// TIA Portal V17 export
// export: Created 2024-08-26T21:07:15.6305429Z, ExportSetting WithDefaults, DisplayName Totally Integrated Automation Portal, DisplayVersion V17 Update 7, DisplayName TIA Portal Openness, DisplayVersion V17 Update 7, DisplayName TIA Portal Version Control Interface, DisplayVersion V17, DisplayName SINAMICS Startdrive Advanced, DisplayVersion V17 SP2, DisplayName SINAMICS Startdrive G110M, G120, G120C, G120D, G120P, G115D, DisplayVersion V17 SP2, DisplayName SINAMICS Startdrive G130, G150, S120, S150, SINAMICS MV, S210, DisplayVersion V17 SP2, DisplayName STEP 7 Professional, DisplayVersion V17 Update 7, DisplayName STEP 7 Safety, DisplayVersion V17 Update 6, DisplayName WinCC Advanced / Unified PC, DisplayVersion V17 Update 7
DATA_BLOCK "DB_INPUTS"   // DB1
{ S7_Optimized_Access := 'TRUE' }
VERSION : 0.1
// stored: AutoNumber false, DBAccessibleFromOPCUA true, DBAccessibleFromWebserver true, IsOnlyStoredInLoadMemory false, IsRetainMemResEnabled false, IsWriteProtectedInAS false, MemoryReserve 100
   VAR RETAIN
      intputSequence : Array[0..32, 0..25] of DInt;   // 32 entradas [modelo, paso]
   END_VAR
   VAR
      activeInputsReq : Array[0..31] of Bool;
   END_VAR
   VAR RETAIN
      maskSequence : Array[0..32, 0..25] of DInt;   // Máscara de entradas
   END_VAR
   VAR
      activeMask : Array[0..31] of Bool;
   END_VAR
   VAR RETAIN
      inputText : Array[0..31] of String;   // Texto HMI de cada entrada
   END_VAR
   VAR
      buttonStatus : Array[0..63] of Bool;
      activeInputsReqDInt : DInt := -2_130_444_284;   // Estado de sensores en directo
      inputActive : Array[0..31] of Bool;
      euchnerReading : Array[0..254] of Char;
      nestScannerReading : String := '';
      upperScannerReading : String := '';
      nestScanerReceived : Array[0..254] of Char;
      nestScanerReceivedString : String := '';
      upperScannerReceived : Array[0..254] of Char;
      upperScannerReceivedString : String := '';
      euchnerReadingString : String := '$01';
      laserReading : Word := 16#0000;
      laserConstant : Real := 0.0005802801;
      laserReadingInt : DInt := 0;
      readingConversion : LReal := 0.0;
      euchnerName : String := '';
      euchner : Array[0..257] of Byte;
   END_VAR
BEGIN
   intputSequence[0,0] := -2_130_444_283;
   intputSequence[0,1] := -1_996_150_012;
   intputSequence[0,2..4] := -2_146_096_376;
   intputSequence[0,5] := -2_130_367_736;
   intputSequence[0,6..7] := -2_130_367_740;
   intputSequence[0,8] := -2_130_444_284;
   intputSequence[0,9..25] := 0;
   intputSequence[1,0] := -2_130_444_283;
   intputSequence[1,1] := -1_996_082_428;
   intputSequence[1,2..3] := -2_142_358_768;
   intputSequence[1,4] := -2_142_358_640;
   intputSequence[1,5] := -2_142_358_652;
   intputSequence[1,6..7] := -2_130_300_156;
   intputSequence[1,8] := -2_130_444_284;
   intputSequence[1,9..25] := 0;
   intputSequence[2,0] := -2_130_444_283;
   intputSequence[2,1] := -1_996_150_012;
   intputSequence[2,2..4] := -2_146_096_376;
   intputSequence[2,5] := -2_130_367_736;
   intputSequence[2,6..7] := -2_130_367_740;
   intputSequence[2,8] := -2_130_444_284;
   intputSequence[2,9..25] := 0;
   intputSequence[3,0] := 84148229;
   intputSequence[3,1] := 1_057_235_716;
   intputSequence[3,2] := 1_175_724_802;
   intputSequence[3,3] := 101_720_834;
   intputSequence[3,4] := 101_982_978;
   intputSequence[3,5] := 84157188;
   intputSequence[3,6] := 84148228;
   intputSequence[3,7..25] := 0;
   intputSequence[4,0] := 84148229;
   intputSequence[4,1] := 1_057_236_740;
   intputSequence[4,2] := 1_175_725_826;
   intputSequence[4,3] := 101_721_858;
   intputSequence[4,4] := 101_984_002;
   intputSequence[4,5] := 84158212;
   intputSequence[4,6] := 84148228;
   intputSequence[4,7..25] := 0;
   intputSequence[5,0] := 84148229;
   intputSequence[5,1] := 1_057_284_868;
   intputSequence[5,2] := 1_175_773_954;
   intputSequence[5,3] := 101_769_986;
   intputSequence[5,4] := 102_032_130;
   intputSequence[5,5] := 84206340;
   intputSequence[5,6] := 84148228;
   intputSequence[5,7..25] := 0;
   intputSequence[6,0] := 84148229;
   intputSequence[6,1] := 1_057_285_892;
   intputSequence[6,2] := 1_175_774_978;
   intputSequence[6,3] := 101_771_010;
   intputSequence[6,4] := 102_033_154;
   intputSequence[6,5] := 84207364;
   intputSequence[6,6] := 84148228;
   intputSequence[6,7..25] := 0;
   intputSequence[7,0] := 23724868;
   intputSequence[7,1] := 827_780_422;
   intputSequence[7,2] := 44756294;
   intputSequence[7,3] := 44755974;
   intputSequence[7,4] := 1_252_650_334;
   intputSequence[7,5..7] := 1_118_432_670;
   intputSequence[7,8] := 1_118_432_414;
   intputSequence[7,9] := 44630336;
   intputSequence[7,10..25] := 0;
   intputSequence[8,0] := 23724353;
   intputSequence[8,1] := 827_776_326;
   intputSequence[8,2] := 44752198;
   intputSequence[8,3] := 44751878;
   intputSequence[8,4] := 1_252_646_238;
   intputSequence[8,5] := 1_118_428_574;
   intputSequence[8,6] := 1_118_428_318;
   intputSequence[8,7] := 1_118_428_574;
   intputSequence[8,8] := 1_118_428_318;
   intputSequence[8,9] := 44630336;
   intputSequence[8,10..25] := 0;
   intputSequence[9,0] := 321;
   intputSequence[9,1] := 4193656;
   intputSequence[9,2] := 2_017_459_576;
   intputSequence[9,3] := 1_077_935_482;
   intputSequence[9,4] := 1_073_745_282;
   intputSequence[9,5..6] := 1_073_745_538;
   intputSequence[9,7..9] := 320;
   intputSequence[9,10..25] := 0;
   intputSequence[10,0] := 321;
   intputSequence[10,1] := 4193656;
   intputSequence[10,2] := 2_017_459_576;
   intputSequence[10,3] := 1_077_935_482;
   intputSequence[10,4] := 1_073_745_282;
   intputSequence[10,5..6] := 1_073_745_538;
   intputSequence[10,7..9] := 320;
   intputSequence[10,10..25] := 0;
   intputSequence[11,0] := 321;
   intputSequence[11,1] := 4193656;
   intputSequence[11,2] := 2_017_459_576;
   intputSequence[11,3] := 1_077_935_482;
   intputSequence[11,4] := 1_073_745_282;
   intputSequence[11,5..6] := 1_073_745_538;
   intputSequence[11,7..9] := 320;
   intputSequence[11,10..25] := 0;
   intputSequence[12,0] := 321;
   intputSequence[12,1] := 8387960;
   intputSequence[12,2] := 2_021_653_880;
   intputSequence[12,3] := 1_082_129_786;
   intputSequence[12,4] := 1_077_939_586;
   intputSequence[12,5] := 1_077_939_842;
   intputSequence[12,6] := 1_073_745_538;
   intputSequence[12,7..9] := 320;
   intputSequence[12,10..25] := 0;
   intputSequence[13,0] := 321;
   intputSequence[13,1] := 4193656;
   intputSequence[13,2] := 2_017_459_576;
   intputSequence[13,3] := 1_077_935_482;
   intputSequence[13,4] := 1_073_745_282;
   intputSequence[13,5..6] := 1_073_745_538;
   intputSequence[13,7..9] := 320;
   intputSequence[13,10..25] := 0;
   intputSequence[14,0] := 321;
   intputSequence[14,1] := 4193656;
   intputSequence[14,2] := 2_017_459_576;
   intputSequence[14,3] := 1_077_935_482;
   intputSequence[14,4] := 1_073_745_282;
   intputSequence[14,5..6] := 1_073_745_538;
   intputSequence[14,7..9] := 320;
   intputSequence[14,10..25] := 0;
   intputSequence[15,0] := 11;
   intputSequence[15,1] := 63040522;
   intputSequence[15,2] := 1_338_108_938;
   intputSequence[15,3] := 65137674;
   intputSequence[15,4] := 65135628;
   intputSequence[15,5] := 65134612;
   intputSequence[15,6] := 57344;
   intputSequence[15,7] := 805_363_712;
   intputSequence[15,8] := 10;
   intputSequence[15,9..25] := 0;
   intputSequence[16,0] := 321;
   intputSequence[16,1] := 8387960;
   intputSequence[16,2] := 2_021_653_880;
   intputSequence[16,3] := 1_082_129_786;
   intputSequence[16,4] := 1_077_939_586;
   intputSequence[16,5] := 1_077_939_842;
   intputSequence[16,6] := 1_073_745_538;
   intputSequence[16,7..9] := 320;
   intputSequence[16,10..25] := 0;
   intputSequence[17,0] := 321;
   intputSequence[17,1] := 4193656;
   intputSequence[17,2] := 2_017_459_576;
   intputSequence[17,3] := 1_077_935_482;
   intputSequence[17,4] := 1_073_745_282;
   intputSequence[17,5..6] := 1_073_745_538;
   intputSequence[17,7..9] := 320;
   intputSequence[17,10..25] := 0;
   intputSequence[18,0] := 321;
   intputSequence[18,1] := 4193656;
   intputSequence[18,2] := 2_017_459_576;
   intputSequence[18,3] := 1_077_935_482;
   intputSequence[18,4] := 1_073_745_282;
   intputSequence[18,5..6] := 1_073_745_538;
   intputSequence[18,7..9] := 320;
   intputSequence[18,10..25] := 0;
   intputSequence[19,0] := 321;
   intputSequence[19,1] := 4193656;
   intputSequence[19,2] := 2_017_459_576;
   intputSequence[19,3] := 1_077_935_482;
   intputSequence[19,4] := 1_073_745_282;
   intputSequence[19,5..6] := 1_073_745_538;
   intputSequence[19,7..9] := 320;
   intputSequence[19,10..25] := 0;
   intputSequence[20,0..25] := 0;
   intputSequence[21,0..25] := 0;
   intputSequence[22,0..25] := 0;
   intputSequence[23,0..25] := 0;
   intputSequence[24,0..25] := 0;
   intputSequence[25,0..25] := 0;
   intputSequence[26,0..25] := 0;
   intputSequence[27,0..25] := 0;
   intputSequence[28,0..25] := 0;
   intputSequence[29,0..25] := 0;
   intputSequence[30,0..25] := 0;
   intputSequence[31,0..25] := 0;
   intputSequence[32,0..25] := 0;
   activeInputsReq[0] := TRUE;
   activeInputsReq[1] := FALSE;
   activeInputsReq[2] := TRUE;
   activeInputsReq[3..17] := FALSE;
   activeInputsReq[18] := TRUE;
   activeInputsReq[19..23] := FALSE;
   activeInputsReq[24] := TRUE;
   activeInputsReq[25..30] := FALSE;
   activeInputsReq[31] := TRUE;
   maskSequence[0,0] := 0;
   maskSequence[0,1] := 805_306_368;
   maskSequence[0,2] := 939_528_320;
   maskSequence[0,3] := 134_221_952;
   maskSequence[0,4] := 146_804_928;
   maskSequence[0,5] := 134_217_856;
   maskSequence[0,6..8] := 134_217_728;
   maskSequence[0,9..25] := 0;
   maskSequence[1,0] := 0;
   maskSequence[1,1] := 805_306_368;
   maskSequence[1,2] := 939_526_144;
   maskSequence[1,3..4] := 134_219_776;
   maskSequence[1,5] := 138_412_160;
   maskSequence[1,6] := 134_221_952;
   maskSequence[1,7..8] := 134_217_728;
   maskSequence[1,9..25] := 0;
   maskSequence[2,0] := 0;
   maskSequence[2,1] := 805_306_368;
   maskSequence[2,2] := 939_528_320;
   maskSequence[2,3] := 134_221_952;
   maskSequence[2,4] := 146_804_928;
   maskSequence[2,5] := 134_217_856;
   maskSequence[2,6..8] := 134_217_728;
   maskSequence[2,9..25] := 0;
   maskSequence[3,0] := 0;
   maskSequence[3,1] := 202752;
   maskSequence[3,2] := 948_115_456;
   maskSequence[3,3] := 2_055_411_712;
   maskSequence[3,4] := 998_447_104;
   maskSequence[3,5] := 948_115_456;
   maskSequence[3,6] := 939_726_848;
   maskSequence[3,7..25] := 0;
   maskSequence[4,0] := 0;
   maskSequence[4,1] := 202752;
   maskSequence[4,2] := 948_115_456;
   maskSequence[4,3] := 2_055_411_712;
   maskSequence[4,4] := 998_447_104;
   maskSequence[4,5] := 948_115_456;
   maskSequence[4,6] := 939_726_848;
   maskSequence[4,7..25] := 0;
   maskSequence[5,0] := 0;
   maskSequence[5,1] := 202752;
   maskSequence[5,2] := 948_115_456;
   maskSequence[5,3] := 2_055_411_712;
   maskSequence[5,4] := 998_447_104;
   maskSequence[5,5] := 948_115_456;
   maskSequence[5,6] := 939_726_848;
   maskSequence[5,7..25] := 0;
   maskSequence[6,0] := 0;
   maskSequence[6,1] := 202752;
   maskSequence[6,2] := 948_115_456;
   maskSequence[6,3] := 2_055_411_712;
   maskSequence[6,4] := 998_447_104;
   maskSequence[6,5] := 948_115_456;
   maskSequence[6,6] := 939_726_848;
   maskSequence[6,7..25] := 0;
   maskSequence[7,0] := 66848767;
   maskSequence[7,1] := 66846720;
   maskSequence[7,2..3] := 66847168;
   maskSequence[7,4..6] := 66846720;
   maskSequence[7,7] := 66846976;
   maskSequence[7,8] := 66846720;
   maskSequence[7,9] := 66847168;
   maskSequence[7,10..25] := 0;
   maskSequence[8,0..1] := 66846720;
   maskSequence[8,2..3] := 66847168;
   maskSequence[8,4..5] := 66846720;
   maskSequence[8,6..7] := 66846976;
   maskSequence[8,8] := 66846720;
   maskSequence[8,9] := 66847168;
   maskSequence[8,10..25] := 0;
   maskSequence[9,0] := -322;
   maskSequence[9,1] := 2_014_248_960;
   maskSequence[9,2..3] := 983040;
   maskSequence[9,4..5] := 79687736;
   maskSequence[9,6] := 134_213_948;
   maskSequence[9,7..8] := -2;
   maskSequence[9,9] := 134_217_406;
   maskSequence[9,10..25] := 0;
   maskSequence[10,0] := -322;
   maskSequence[10,1] := 2_014_289_920;
   maskSequence[10,2..3] := 1024000;
   maskSequence[10,4..5] := 79687736;
   maskSequence[10,6] := 134_213_948;
   maskSequence[10,7..8] := -2;
   maskSequence[10,9] := 134_217_406;
   maskSequence[10,10..25] := 0;
   maskSequence[11,0] := -322;
   maskSequence[11,1] := 2_014_248_960;
   maskSequence[11,2..3] := 983040;
   maskSequence[11,4..5] := 79687736;
   maskSequence[11,6] := 134_213_948;
   maskSequence[11,7..8] := -2;
   maskSequence[11,9] := 134_217_406;
   maskSequence[11,10..25] := 0;
   maskSequence[12,0] := -322;
   maskSequence[12,1] := 2_014_248_960;
   maskSequence[12,2..3] := 983040;
   maskSequence[12,4..5] := 79687736;
   maskSequence[12,6] := 134_213_948;
   maskSequence[12,7..8] := -2;
   maskSequence[12,9] := 134_217_406;
   maskSequence[12,10..25] := 0;
   maskSequence[13,0] := -322;
   maskSequence[13,1] := 2_014_248_960;
   maskSequence[13,2..3] := 983040;
   maskSequence[13,4..5] := 79687736;
   maskSequence[13,6] := 134_213_948;
   maskSequence[13,7..8] := -2;
   maskSequence[13,9] := 134_217_406;
   maskSequence[13,10..25] := 0;
   maskSequence[14,0] := -322;
   maskSequence[14,1] := 2_014_248_960;
   maskSequence[14,2] := 806_289_408;
   maskSequence[14,3] := 983040;
   maskSequence[14,4..5] := 79687736;
   maskSequence[14,6] := 134_213_948;
   maskSequence[14,7..8] := -2;
   maskSequence[14,9] := 134_217_406;
   maskSequence[14,10..25] := 0;
   maskSequence[15,0] := 0;
   maskSequence[15,1] := 2_080_374_784;
   maskSequence[15,2..3] := 805_306_368;
   maskSequence[15,4..5] := 868_220_928;
   maskSequence[15,6..7] := 268_435_452;
   maskSequence[15,8..25] := 0;
   maskSequence[16,0] := -322;
   maskSequence[16,1] := 2_014_248_960;
   maskSequence[16,2..3] := 983040;
   maskSequence[16,4..5] := 79687736;
   maskSequence[16,6] := 134_213_948;
   maskSequence[16,7..8] := -2;
   maskSequence[16,9] := 134_217_406;
   maskSequence[16,10..25] := 0;
   maskSequence[17,0] := -322;
   maskSequence[17,1] := 2_014_248_960;
   maskSequence[17,2..3] := 983040;
   maskSequence[17,4..5] := 79687736;
   maskSequence[17,6] := 134_213_948;
   maskSequence[17,7..8] := -2;
   maskSequence[17,9] := 134_217_406;
   maskSequence[17,10..25] := 0;
   maskSequence[18,0] := -322;
   maskSequence[18,1] := 2_014_248_960;
   maskSequence[18,2..3] := 983040;
   maskSequence[18,4..5] := 79687736;
   maskSequence[18,6] := 134_213_948;
   maskSequence[18,7..8] := -2;
   maskSequence[18,9] := 134_217_406;
   maskSequence[18,10..25] := 0;
   maskSequence[19,0] := -322;
   maskSequence[19,1] := 2_014_248_960;
   maskSequence[19,2..3] := 983040;
   maskSequence[19,4..5] := 79687736;
   maskSequence[19,6] := 134_213_948;
   maskSequence[19,7..8] := -2;
   maskSequence[19,9] := 134_217_406;
   maskSequence[19,10..25] := 0;
   maskSequence[20,0..25] := 0;
   maskSequence[21,0..25] := 0;
   maskSequence[22,0..25] := 0;
   maskSequence[23,0..25] := 0;
   maskSequence[24,0..25] := 0;
   maskSequence[25,0..25] := 0;
   maskSequence[26,0..25] := 0;
   maskSequence[27,0..25] := 0;
   maskSequence[28,0..25] := 0;
   maskSequence[29,0..25] := 0;
   maskSequence[30,0..25] := 0;
   maskSequence[31,0..25] := 0;
   maskSequence[32,0..25] := 0;
   activeMask[0..31] := FALSE;
   inputText[0] := 'CLEAR DATA';
   inputText[1] := 'LEFT TOOLING WORK POS';
   inputText[2] := 'LEFTTOOLING HOME POS';
   inputText[3] := 'LEFT TOOLING POS 1';
   inputText[4] := 'LEFT TOOOLLING POS 3';
   inputText[5] := 'LEFT TOOLING POS 2';
   inputText[6] := 'LEFT INSERTIONN EXT NOK';
   inputText[7] := 'LEFT INSERTIONN EXT OK';
   inputText[8] := 'PRODUCT INSERTED LH';
   inputText[9] := 'PRODUCT INSERTED RH';
   inputText[10] := 'STRAP DETECTION';
   inputText[11] := 'LEFT MANUAL FRAME PRES';
   inputText[12] := 'RIGHT MANUAL FRAME PRES';
   inputText[13] := 'FRAME PRES';
   inputText[14] := 'LEFTT BRACKET DETECTION';
   inputText[15] := 'RIGHT BRACKET DETECTION';
   inputText[16] := 'LEFT COLOR SPRING';
   inputText[17] := 'RIGHT COLOR SPRING';
   inputText[18] := 'TORQUE TOOLING HOME';
   inputText[19] := 'RIGHT TOOLING POS 1';
   inputText[20] := 'RIGHT TOOLING POS 3';
   inputText[21] := 'RIGHT TOOLING POS 2';
   inputText[22] := 'RIGHT INSERTION EXT OK';
   inputText[23] := 'RIGHT INSERTION EXTNOK';
   inputText[24] := 'RIGHT TOOLING HOME';
   inputText[25] := 'WASHER INSERTED';
   inputText[26] := 'POWER TOOLING';
   inputText[27] := 'NEST SCANNER';
   inputText[28] := 'ANGLE SCANNER';
   inputText[29] := 'UPPER SCANNER LABEL1';
   inputText[30] := 'UPPER SCANNER LABEL 2';
   inputText[31] := 'MANUAL TOOLING';
   buttonStatus[0..2] := FALSE;
   buttonStatus[3] := TRUE;
   buttonStatus[4..7] := FALSE;
   buttonStatus[8..9] := TRUE;
   buttonStatus[10] := FALSE;
   buttonStatus[11] := TRUE;
   buttonStatus[12] := FALSE;
   buttonStatus[13] := TRUE;
   buttonStatus[14..15] := FALSE;
   buttonStatus[16] := TRUE;
   buttonStatus[17] := FALSE;
   buttonStatus[18] := TRUE;
   buttonStatus[19] := FALSE;
   buttonStatus[20] := TRUE;
   buttonStatus[21..30] := FALSE;
   buttonStatus[31] := TRUE;
   buttonStatus[32..38] := FALSE;
   buttonStatus[39] := TRUE;
   buttonStatus[40..43] := FALSE;
   buttonStatus[44] := TRUE;
   buttonStatus[45..58] := FALSE;
   buttonStatus[59] := TRUE;
   buttonStatus[60..63] := FALSE;
   inputActive[0..1] := FALSE;
   inputActive[2] := TRUE;
   inputActive[3..7] := FALSE;
   inputActive[8..9] := TRUE;
   inputActive[10] := FALSE;
   inputActive[11..13] := TRUE;
   inputActive[14..16] := FALSE;
   inputActive[17..18] := TRUE;
   inputActive[19..23] := FALSE;
   inputActive[24] := TRUE;
   inputActive[25..30] := FALSE;
   inputActive[31] := TRUE;
   euchnerReading[0] := '$01';
   euchnerReading[1..127] := '$00';
   euchnerReading[128..254] := ' ';
   nestScanerReceived[0..254] := ' ';
   upperScannerReceived[0..254] := ' ';
   euchner[0..1] := 16#00;
   euchner[2] := 16#44;
   euchner[3..7] := 16#00;
   euchner[8..147] := 16#20;
   euchner[148..257] := 16#00;
END_DATA_BLOCK
